// TIA Portal V18 export
DATA_BLOCK "ROBOT_DATA_DB"   // DB5
{ S7_Optimized_Access := 'FALSE' }
   VAR
      INPUT : "RBT_TO_PLC";
      OUTPUT : "PLC_TO_RBT";
   END_VAR
BEGIN
END_DATA_BLOCK
